FUNCTION_BLOCK Axis_Limit_Stop
VAR_INPUT
	Execute_:BOOL;
	Execute_2:BOOL;
	Decelerations: INT;
END_VAR
VAR_OUTPUT
	Flag1:BOOL;
	Flag2:BOOL;
END_VAR
VAR
	AxisStop:MC_Stop;
	trig1: F_TRIG;
END_VAR

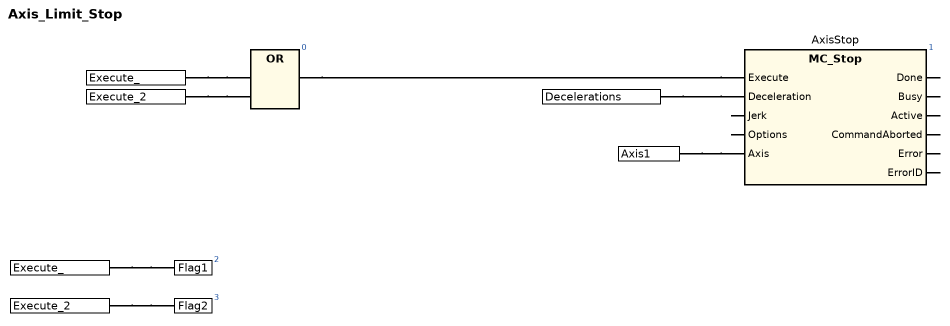
AxisStop(Execute := Execute_ OR Execute_2, Deceleration := Decelerations, Axis := Axis1); // MC_Stop
Flag1 := Execute_;
Flag2 := Execute_2;

END_FUNCTION_BLOCK

(* stored: Version 1.1.0.1, ProductVersion 3.1.4024.12
   POU Axis_Limit_Stop: Id {0666d1dc-d921-4672-84d8-e2867a267642}, SpecialFunc None *)
